Staubli VAL3: prdStatusList.pgx

program prdStatusList()
  local num l_nI
  local string l_sSBuff
  local bool l_bBool
  local string l_sItems
begin
  //生产状态栏

  //2015.02.02
  call use:setSizeList(20,0,18,10)
  call use:listcreate("状态列表")

  sPrdStatus[0]="Txt文件:"
  if len(sTxtSelected)==0
    sPrdStatus[1]="未选择"
  else
    sPrdStatus[1]=sTxtSelected
  endIf
  if read:bCycle==false
    if bSuspend
      sPrdStatus[2]="生产状态:"+"等待复位"
    else
      sPrdStatus[2]="生产状态:"+"无生产"
    endIf
  elseIf bPause==true
    sPrdStatus[2]="生产状态:"+"暂停中"
  else
    sPrdStatus[2]="生产状态:"+"生产中"
  endIf
  if nWorkModeStatus==2
    sPrdStatus[3]="运动状态:"+"Hold"
  else
    sPrdStatus[3]="运动状态:"+"Move"
  endIf
  sPrdStatus[4]="总路径个数:"+toString("6.0",read:nTotalTrajs)
  sPrdStatus[5]="当前路径  :"+toString("6.0",read:nTrajofRead+1)
  sPrdStatus[6]="写入点个数:"+toString("6.0",read:nWritePtr+read:nThousandWrite*1000)
  sPrdStatus[7]="读取点个数:"+toString("6.0",read:nReadPtr+read:nThousandRead*1000)
  sPrdStatus[8]="当前MoveID:"+toString("6.0",read:nMoveID)
  sPrdStatus[9]="瞬时速度  :"+toString("6.2",read:nSpdOfTCP)

  //2015.02.02
  call use:listadd(sPrdStatus)
  call use:listupdate1(0)

  if l_sSBuff!=sPrdStatus[2]

    //  call UI:Control_PanelMd(sPrdStatus[2])
    l_sSBuff=sPrdStatus
    if bPause
      l_sItems=",启动,继续,停止,,回零,,退出"
    else
      l_sItems=",启动,暂停,停止,,回零,,退出"
    endIf
    call use:stringToArray(l_sItems,sItems)
    call use:setMenu(sItems,true,3)
    // call UI:Form_Prod(sItems)
    //call UI:Control_Bottom(sItems)
  endIf

  //  if l_bBool!=bPause
  //
  //    // call UI:Control_PanelMd(sPrdStatus[2])
  //    l_bBool=bPause
  //  endIf

  gotoxy(0,11)
  //put("间断时长:"+toString(".1",nPauseTime)+"秒")


end
